// TIA Portal V21 export
TYPE "LAxisCtrl_typeHoming"
TITLE = LAxisCtrl_typeHoming
// Support: tech.team.motioncontrol@siemens.com
   STRUCT
      position : LReal := 0.0;   // The specified value is used according to the selected "Mode"
      mode : Int := 0;   // Operation mode; 0: Direct homing (absolute); 1: Direct homing (relative); 2: Passive homing (without reset); 3: Active homing; 5: Active homing (Position parameter has no effect); 6: Absolute encoder adjustment (relative); 7: Absolute encoder adjustment (absolute); 8: Passive homing; 9: Abort passive homing; 10: Passive homing (Position parameter has no effect); 11: Set setpoint position (absolute); 12: Shift the setpoint position (relative); 13: Incremental encoder adjustment
      sensor : DInt := 0;   // Only relevant for S7-1500T: Selection of the absolute encoder ("Mode" = 6, 7) or incremental encoder ("Mode" = 13) to be calibrated; 0: Operative encoder; 1..4: Encoder 1..4 (S7-1500T)
      extendedMode : DInt := -1;   // -1: No extended homing mode (parameter "mode" is effective); 0: Homing on fixed stop; 1: Homing on fixed stop with moving out of clamping; 2: Homing on fixed stop with moving to target position
      extendedModeTorqueLimit : LReal := 0.0;   // Value of the torque/force for extended homing mode
      extendedModeTargetPosition : LReal := 0.0;   // Target position when 'extendedMode' = 2
   END_STRUCT;
END_TYPE
